{attribute 'linkalways'} 
{attribute 'no_explicit_call' := 'This FB is a CLASS and must be accessed using methods or properties'}
{attribute 'enable_dynamic_creation'}
FUNCTION_BLOCK FINAL AND_DINT EXTENDS Node
VAR
	in1 : _DINT(0);
	in2 : _DINT(0);
	out : _DINT(0);
END_VAR

METHOD PUBLIC Clone : I_Node
VAR
	pNode : POINTER TO AND_DINT;
END_VAR
pNode := __NEW(AND_DINT);
Clone := pNode^;
END_METHOD

METHOD FB_init : BOOL
VAR_INPUT
	bInitRetains : BOOL; // if TRUE, the retain variables are initialized (warm start / cold start)
	bInCopyCode : BOOL;  // if TRUE, the instance afterwards gets moved into the copy code (online change)
END_VAR
AddInput('in1',THIS^.in1);
AddInput('in2',THIS^.in2);
AddOutput('out', THIS^.out);
END_METHOD

METHOD PROTECTED OnExecute
VAR
END_VAR
out.Value := in1.Value AND in2.Value;
END_METHOD

END_FUNCTION_BLOCK

(* stored: Version 1.1.0.1, ProductVersion 3.1.4024.15
   POU AND_DINT: Id {96aebf06-acf7-4a44-b339-0a5ebdbeec66}, SpecialFunc None
   Folder Constructor: Id {10e602a8-7a17-402a-84c9-e774be0b1b9f}
   Method Clone: Id {f18718c3-08e5-4fa2-a40d-a2afcf65054f}
   Method FB_init: Id {56e24e12-238f-4a70-b939-fd06ed5c160b}
   Method OnExecute: Id {8f9a51c1-e6b1-470c-8d92-dfe45c74e2c9} *)
